FUNCTION_BLOCK FB_KVM
VAR_INPUT
	wAID: WORD;
END_VAR
VAR_OUTPUT
END_VAR
VAR
	fbTonLive: TON;
	ftriboSystemResetBut: F_TRIG;
END_VAR

IF fbTonLive.Q THEN	KVM.gstKVM.stStatus.boLive:=NOT KVM.gstKVM.stStatus.boLive; END_IF
fbTonLive(IN:=NOT fbTonLive.Q , PT:=T#500MS , Q=> , ET=> );

// AID - Application ID
KVM.gstKVM.stApp.wAID:=wAID;

// selection of application
IF 		wAID=1 THEN	App1();
ELSIF 	wAID=2 THEN	App2(); END_IF

Safety();
General();

ACTION App1:
KVM.gstKVM.stApp.sName:='Cartesian Application';
KVM.gstKVM.stApp.sInfo:='Pick $R$Nand place';


KVM.gstKVM.stCA.lrCA[0]:=Axis.stAxis1.NcToPlc.ActPos;
KVM.gstKVM.stCA.lrCA[1]:=Axis.stAxis2.NcToPlc.ActPos;
KVM.gstKVM.stCA.lrCA[2]:=Axis.stAxis3.NcToPlc.ActPos;
END_ACTION

ACTION App2:
;
END_ACTION

ACTION General:

// status
KVM.gstKVM.stStatus.lrElapsedTimeSec:=KVM.gstKVM.stStatus.lrElapsedTimeSec+KVM.lrCycleSec;

// inputs
INPUT.iboIN0_EmergencyStopBut:=KVM.gstKVM.stAC.boAC[0];			KVM.gstKVM.stAC.sboACComments[0]:='Emergency button';
INPUT.iboIN1_StartBut:=KVM.gstKVM.stAC.boAC[1];					KVM.gstKVM.stAC.sboACComments[1]:='Start button';
INPUT.iboIN2_StopBut:=KVM.gstKVM.stAC.boAC[2];					KVM.gstKVM.stAC.sboACComments[2]:='Stop button';
INPUT.iboIN3_AlarmResetBut:=KVM.gstKVM.stAC.boAC[3];			KVM.gstKVM.stAC.sboACComments[3]:='Alarm reset button';
INPUT.iboIN4_SystemResetBut:=KVM.gstKVM.stAC.boAC[4];			KVM.gstKVM.stAC.sboACComments[4]:='System reset button';
INPUT.iboIN5_AutoBut:=KVM.gstKVM.stAC.boAC[5];					KVM.gstKVM.stAC.sboACComments[5]:='Auto / man button';
INPUT.iboIN6_PauseBut:=KVM.gstKVM.stAC.boAC[6];					KVM.gstKVM.stAC.sboACComments[6]:='Pause button';
INPUT.iboIN7_StepBut:=KVM.gstKVM.stAC.boAC[7];					KVM.gstKVM.stAC.sboACComments[7]:='Step button';
                                                        	
INPUT.iboIN8_ManFwdBut:=KVM.gstKVM.stAC.boAC[8];				KVM.gstKVM.stAC.sboACComments[8]:='Man forward button';
INPUT.iboIN9_ManBwdBut:=KVM.gstKVM.stAC.boAC[9];				KVM.gstKVM.stAC.sboACComments[9]:='Man backward button';
(**)                                                    	
(**)                                                    	
(**)                                                    	
(**)                                                    	
(**)                                                    	
(**)                                                    	
                                                        	
INPUT.iboIN16_Axis1PosLimSw:=KVM.gstKVM.stAC.boAC[16];			KVM.gstKVM.stAC.sboACComments[16]:='Axis 1 of pos. limit switch';
INPUT.iboIN17_Axis1NegLimSw:=KVM.gstKVM.stAC.boAC[17];			KVM.gstKVM.stAC.sboACComments[17]:='Axis 1 of neg. limit switch';
INPUT.iboIN18_Axis2PosLimSw:=KVM.gstKVM.stAC.boAC[18];			KVM.gstKVM.stAC.sboACComments[18]:='Axis 2 of pos. limit switch';
INPUT.iboIN19_Axis2NegLimSw:=KVM.gstKVM.stAC.boAC[19];			KVM.gstKVM.stAC.sboACComments[19]:='Axis 2 of neg. limit switch';
INPUT.iboIN20_Axis3PosLimSw:=KVM.gstKVM.stAC.boAC[20];			KVM.gstKVM.stAC.sboACComments[20]:='Axis 3 of pos. limit switch';
INPUT.iboIN21_Axis3NegLimSw:=KVM.gstKVM.stAC.boAC[21];			KVM.gstKVM.stAC.sboACComments[21]:='Axis 3 of neg. limit switch';
INPUT.iboIN22_Axis4PosLimSw:=KVM.gstKVM.stAC.boAC[22];			KVM.gstKVM.stAC.sboACComments[22]:='Axis 4 of pos. limit switch';
INPUT.iboIN23_Axis4NegLimSw:=KVM.gstKVM.stAC.boAC[23];			KVM.gstKVM.stAC.sboACComments[23]:='Axis 4 of neg. limit switch';



// outputs
KVM.gstKVM.stCA.boCA[0]:=OUTPUT.qboOUT0_STO;					KVM.gstKVM.stCA.sboCAComments[0]:='Safe torque off';
KVM.gstKVM.stCA.boCA[1]:=OUTPUT.qboOUT1_StartLam;				KVM.gstKVM.stCA.sboCAComments[1]:='Lamp of start button';
KVM.gstKVM.stCA.boCA[2]:=OUTPUT.qboOUT2_StopLam;				KVM.gstKVM.stCA.sboCAComments[2]:='Lamp of stop button';
KVM.gstKVM.stCA.boCA[3]:=OUTPUT.qboOUT3_AlarmLam;				KVM.gstKVM.stCA.sboCAComments[3]:='Lamp of alarm';
KVM.gstKVM.stCA.boCA[4]:=OUTPUT.qboOUT4_SystemLam;				KVM.gstKVM.stCA.sboCAComments[4]:='Lamp of safety';
KVM.gstKVM.stCA.boCA[5]:=OUTPUT.qboOUT5_AutoLam;				KVM.gstKVM.stCA.sboCAComments[5]:='Lamp of auto button';
KVM.gstKVM.stCA.boCA[6]:=OUTPUT.qboOUT6_PauseLam;				KVM.gstKVM.stCA.sboCAComments[6]:='Lamp of pause button';
KVM.gstKVM.stCA.boCA[7]:=OUTPUT.qboOUT7_StepLam;				KVM.gstKVM.stCA.sboCAComments[7]:='Lamp of step button';

KVM.gstKVM.stCA.boCA[8]:=OUTPUT.qboOUT8_ManFwdLam;				KVM.gstKVM.stCA.sboCAComments[8]:='Lamp of forward button';
KVM.gstKVM.stCA.boCA[9]:=OUTPUT.qboOUT9_ManBwdLam;				KVM.gstKVM.stCA.sboCAComments[9]:='Lamp of backward button';
(**)                                                    	
(**)                                                    	
(**)  
KVM.gstKVM.stCA.boCA[13]:=OUTPUT.qboOUT13_TowerLightRedLam;		KVM.gstKVM.stCA.sboCAComments[13]:='Light tower red lamp';
KVM.gstKVM.stCA.boCA[14]:=OUTPUT.qboOUT14_TowerLightYellowLam;	KVM.gstKVM.stCA.sboCAComments[14]:='Light tower yellow lamp';
KVM.gstKVM.stCA.boCA[15]:=OUTPUT.qboOUT15_TowerLightGreenLam;	KVM.gstKVM.stCA.sboCAComments[15]:='Light tower green lamp';
END_ACTION

ACTION Safety:
ftriboSystemResetBut(CLK:=INPUT.iboIN4_SystemResetBut, Q=>);
IF INPUT.iboIN0_EmergencyStopBut AND ftriboSystemResetBut.Q THEN
	OUTPUT.qboOUT0_STO:=TRUE;
END_IF

IF NOT INPUT.iboIN0_EmergencyStopBut THEN
	OUTPUT.qboOUT0_STO:=FALSE;
END_IF

OUTPUT.qboOUT4_SystemLam:=OUTPUT.qboOUT0_STO OR KVM.gstKVM.stStatus.boLive;
END_ACTION

END_FUNCTION_BLOCK

(* stored: Version 1.1.0.1, ProductVersion 3.1.4024.12
   POU FB_KVM: Id {8b6dbdab-54ad-4655-bd64-d07505511630}, SpecialFunc None
   Action App1: Id {7424dcda-d0f7-4aa2-bed9-d9611ccf6c52}
   Action App2: Id {07759514-4541-4148-8fc8-41dbe14d4891}
   Action General: Id {41bab375-2a83-40cb-b0b0-259fb3913f5a}
   Action Safety: Id {f0e97837-7355-444c-b566-26605a6402c4} *)
